FUNCTION_BLOCK FB_Light
VAR
	licht		AT %Q*	: BOOL;
END_VAR

METHOD Turn_off : BOOL
VAR_INPUT
END_VAR
licht	:= FALSE;
END_METHOD

METHOD Turn_on : BOOL
VAR_INPUT
END_VAR
licht	:= TRUE;
END_METHOD

END_FUNCTION_BLOCK

(* stored: Version 1.1.0.1, ProductVersion 3.1.4024.12
   POU FB_Light: Id {9d175803-8873-46a0-a95d-9215d0d9e0f1}, SpecialFunc None
   Method Turn_off: Id {288dcc40-7e6a-4bda-a2c8-45b15b6f44a5}
   Method Turn_on: Id {9b2bb554-fa6e-4c1e-b69b-a3f60fcd7250} *)
